PROGRAM P_Vision
VAR
	bBlobExecution		:BOOL	:=FALSE;

	bTF7820Execution	:BOOL	:=FALSE;
	bTF3820Execution	:BOOL	:=FALSE;
END_VAR

IF bBlobExecution=TRUE AND bTF7820Execution=FALSE AND bTF3820Execution=FALSE THEN
	P_BlobVision();
ELSIF bBlobExecution=FALSE AND bTF7820Execution=TRUE AND bTF3820Execution=FALSE THEN
	P_DNNVision();
ELSIF bBlobExecution=FALSE and bTF7820Execution=FALSE AND bTF3820Execution=TRUE THEN
	P_MLSVision();
END_IF

END_PROGRAM

(* stored: Version 1.1.0.1, ProductVersion 3.1.4026.18
   POU P_Vision: Id {12aa390b-17e5-4f54-a4d0-60c6f0bb99e7}, SpecialFunc None *)
